// Mitsubishi GX Works2 project: test 1   PLC: FX3U/FX3UC

PROGRAM MAIN
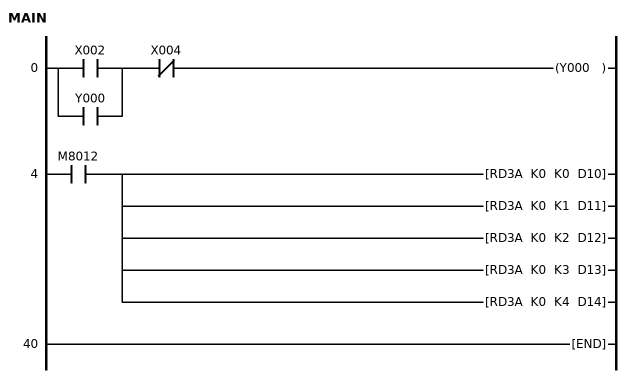
0     LD      X002
      OR      Y000
      ANI     X004
      OUT     Y000
4     LD      M8012
      RD3A    K0 K0 D10
      RD3A    K0 K1 D11
      RD3A    K0 K2 D12
      RD3A    K0 K3 D13
      RD3A    K0 K4 D14
40    END
END_PROGRAM
